Yaskawa INFORM job: WELDING-CMF100-ST2-BACK.JBI

/JOB
//NAME WELDING-CMF100-ST2-BACK
//POS
///NPOS 16,16,16,1,0,0
///TOOL 0
///POSTYPE PULSE
///PULSE
C00000=72547,-33316,-23472,-62404,52759,85582
C00001=64766,-25915,-39604,-94670,51413,102994
C00002=77738,780,-21384,-104658,58925,108021
C00003=77222,36515,-52625,-145994,2143,131014
C00004=77222,36423,-52613,-145993,2195,131003
C00005=77322,36229,-52837,-146054,2161,131032
C00006=78871,3738,-15581,-95747,61329,103014
C00007=78871,3738,-15581,-95747,61329,103014
C00008=78871,3738,-15581,-95747,61329,103014
C00009=78871,3738,-15581,-95747,61329,103014
C00010=110603,52002,77101,3198,24241,47259
C00011=110539,51631,76759,3160,24281,47283
C00012=85688,-2806,-12138,-82418,66697,94466
C00013=70532,-36923,-29307,-69994,55758,87249
C00014=83044,-46385,-33840,-70581,45962,87604
C00015=87141,-40130,-36591,-38139,38419,72570
BC00000=82159
BC00001=74641
BC00002=74641
BC00003=74641
BC00004=74641
BC00005=74641
BC00006=74641
BC00007=74641
BC00008=74641
BC00009=74641
BC00010=131407
BC00011=131407
BC00012=90275
BC00013=90275
BC00014=90275
BC00015=90275
EC00000=2040211
EC00001=2040211
EC00002=2040211
EC00003=2426179
EC00004=2426179
EC00005=2426179
EC00006=2053607
EC00007=1025609
EC00008=17705
EC00009=-1030237
EC00010=-1556687
EC00011=-1556687
EC00012=-1029623
EC00013=-1029623
EC00014=-1029623
EC00015=-665795
///USER 10
///POSTYPE USER
///RECTAN
///RCONF 0,0,0,0,0,0,0,0,0,0,0,0,0,0,0,0,0,0,0,0,0,0,0,0
P00049=2.600,0.000,0.000,0.0000,0.0000,0.0000
//INST
///DATE 2018/10/02 11:25
///ATTR SC,RW
///GROUP1 RB1,BS1
///GROUP2 ST2
NOP
'***** welding station 1 front
MOVJ C00000 BC00000 VJ=25.00  +MOVJ EC00000 VJ=100.00
'***** go to start pos
SMOVL C00001 BC00001 V=166.7 PL=0  +MOVJ EC00001
SMOVL C00002 BC00002 V=83.3  +MOVJ EC00002
SFTON P049 UF#(10)
SMOVC C00003 BC00003 V=83.3 PL=0  +MOVJ EC00003  //start welding
DOUT OT#(656) OFF
TIMER T=0.50
DOUT OT#(656) ON
MACRO1 MJ#(5) ARGF2
SREFP 1 C00004 BC00004  +REFP EC00004
SREFP 2 C00005 BC00005  +REFP EC00005
ARCON ASF#(1)
SWVON WEV#(1)
SMOVC C00006 BC00006 V=I000  +MOVJ EC00006
SMOVC C00007 BC00007 V=I000  +MOVJ EC00007
SMOVC C00008 BC00008 V=I000  +MOVJ EC00008
SMOVC C00009 BC00009 V=I000  +MOVJ EC00009
SMOVC C00010 BC00010 V=I000  +MOVJ EC00010
SMOVC C00011 BC00011 V=I000  +MOVJ EC00011
ARCOF
MACRO1 MJ#(5) ARGF5
DOUT OT#(656) OFF
SWVOF
TIMER T=5.00
'***** go to end position
SFTOF
SMOVL C00012 BC00012 V=16.7 PL=0  +MOVJ EC00012
SMOVL C00013 BC00013 V=83.3  +MOVJ EC00013
SMOVL C00014 BC00014 V=250.0  +MOVJ EC00014
MOVL C00015 BC00015 V=166.7  +MOVJ EC00015 VJ=100.00
END
